// TIA Portal V19 export
TYPE "UnitInitConfig"
// stored: Access Published
   STRUCT
      UnitNo : Int;
   END_STRUCT;
END_TYPE
